// TwinCAT 3 PLC project Plc
// ProgramVersion: 3.1.4023.0
// libraries:
//   Tc2_Standard, * (Beckhoff Automation GmbH)
//   Tc2_System, * (Beckhoff Automation GmbH)
//   Tc3_Module, * (Beckhoff Automation GmbH)
// project tree:
//   / PlcTask.TcTTO (not stored)
//   DUTs/IO/PdoEntries/ Channel_D623F56C.TcDUT
//   DUTs/IO/PDOs/ InfoData_6F19DB2B.TcDUT (not stored), DIG_Outputs_F9744C66.TcDUT, WcState_0B2B16F9.TcDUT, InfoData_32EB74EA.TcDUT, InfoData_E68C61CD.TcDUT (not stored), InfoData_2A97D6CF.TcDUT (not stored), Inputs_A65FACA4.TcDUT (not stored), Outputs_23C0ED1D.TcDUT (not stored)
//   DUTs/IO/Boxes/ EK1100_1FC0878B.TcDUT (not stored), EL2044_DE371F9A.TcDUT
//   DUTs/IO/Devices/ SyncUnitTask_2D604ED5.TcDUT (not stored), SyncUnitTasks_6FEB8257.TcDUT (not stored), SyncUnits_99E584AF.TcDUT (not stored)
//   DUTs/IO/Topology/ Term_1_EK1100_C568EA04.TcDUT (not stored), Device_1_EtherCAT_15E26550.TcDUT (not stored)
//   DUTs/IO/Base/ EtcSlaveBase_82538BE2.TcDUT (not stored), EtcSlaveBase_82538BE2.TcDUT (not stored), EtcSlaveBase_82538BE2.TcDUT (not stored), EtcSlaveTerminalBase_947E5A46.TcDUT (not stored), EtcSlaveBoxBase_77A0E4A7.TcDUT (not stored), EtcSlaveEndTerminalBase_866C7F0C.TcDUT (not stored), InputBase_8311D824.TcDUT (not stored), OutputBase_10CEE7DE.TcDUT (not stored), EtcMasterBase_62654B43.TcDUT (not stored)
//   GVLs/ GVL_iXlinker.TcGVL (not stored)
// real-time tasks:
//   TASK PlcTask: cycle T#10ms, priority 20, ADS port 350
// I/O:
//   DEVICE Device 1 (EtherCAT), AmsNetId 172.20.30.238.2.1
//     Term 1 (EK1100) [EK1100 EtherCAT Coupler (2A E-Bus)]
//       Term 2 (EL2044) [EL2044 4Ch. Dig. Output 24V, 2A, Diagnostic]
// variable links:
//   Plc/Plc Instance <-> Device 1 (EtherCAT)/Term 1 (EK1100)
//     PlcTask Inputs/GVL_iXlinker.Device_1_EtherCAT.Term_1_EK1100.InfoData.State <-> InfoData/State
//   Plc/Plc Instance <-> Device 1 (EtherCAT)/Term 1 (EK1100)/Term 2 (EL2044)
//     PlcTask Outputs/GVL_iXlinker.Device_1_EtherCAT.Term_1_EK1100.Term_2_EL2044.DIG_Outputs.Channel_{1..4}/Output <-> DIG Outputs/Channel {1..4}/Output  (4 links)
//     PlcTask Inputs/GVL_iXlinker.Device_1_EtherCAT.Term_1_EK1100.Term_2_EL2044.WcState.WcState <-> WcState/WcState
//     PlcTask Inputs/GVL_iXlinker.Device_1_EtherCAT.Term_1_EK1100.Term_2_EL2044.InfoData.AdsAddr <-> InfoData/AdsAddr
//     PlcTask Inputs/GVL_iXlinker.Device_1_EtherCAT.Term_1_EK1100.Term_2_EL2044.InfoData.State <-> InfoData/State
//   Plc/Plc Instance <-> Device 1 (EtherCAT)
//     PlcTask Inputs/GVL_iXlinker.Device_1_EtherCAT.SyncUnits._default._unreferenced.WcState.WcState <-> SyncUnits/<default>/<unreferenced>/WcState/WcState
//     PlcTask Inputs/GVL_iXlinker.Device_1_EtherCAT.SyncUnits._default._unreferenced.InfoData.ObjectId <-> SyncUnits/<default>/<unreferenced>/InfoData/ObjectId
//     PlcTask Inputs/GVL_iXlinker.Device_1_EtherCAT.SyncUnits._default._unreferenced.InfoData.State <-> SyncUnits/<default>/<unreferenced>/InfoData/State
//     PlcTask Inputs/GVL_iXlinker.Device_1_EtherCAT.SyncUnits._default._unreferenced.InfoData.SlaveCount <-> SyncUnits/<default>/<unreferenced>/InfoData/SlaveCount
//     PlcTask Inputs/GVL_iXlinker.Device_1_EtherCAT.SyncUnits._default.PlcTask.WcState.WcState <-> SyncUnits/<default>/PlcTask/WcState/WcState
//     PlcTask Inputs/GVL_iXlinker.Device_1_EtherCAT.SyncUnits._default.PlcTask.InfoData.ObjectId <-> SyncUnits/<default>/PlcTask/InfoData/ObjectId
//     PlcTask Inputs/GVL_iXlinker.Device_1_EtherCAT.SyncUnits._default.PlcTask.InfoData.State <-> SyncUnits/<default>/PlcTask/InfoData/State
//     PlcTask Inputs/GVL_iXlinker.Device_1_EtherCAT.SyncUnits._default.PlcTask.InfoData.SlaveCount <-> SyncUnits/<default>/PlcTask/InfoData/SlaveCount
//     PlcTask Inputs/GVL_iXlinker.Device_1_EtherCAT.Inputs.SlaveCount <-> Inputs/SlaveCount
//     PlcTask Inputs/GVL_iXlinker.Device_1_EtherCAT.Inputs.DevState <-> Inputs/DevState
//     PlcTask Inputs/GVL_iXlinker.Device_1_EtherCAT.Inputs.Frm0State <-> Inputs/Frm0State
//     PlcTask Inputs/GVL_iXlinker.Device_1_EtherCAT.Inputs.Frm0WcState <-> Inputs/Frm0WcState
//     PlcTask Inputs/GVL_iXlinker.Device_1_EtherCAT.Inputs.Frm0InputToggle <-> Inputs/Frm0InputToggle
//     PlcTask Outputs/GVL_iXlinker.Device_1_EtherCAT.Outputs.DevCtrl <-> Outputs/DevCtrl
//     PlcTask Outputs/GVL_iXlinker.Device_1_EtherCAT.Outputs.Frm0Ctrl <-> Outputs/Frm0Ctrl
//     PlcTask Outputs/GVL_iXlinker.Device_1_EtherCAT.Outputs.Frm0WcCtrl <-> Outputs/Frm0WcCtrl
//     PlcTask Inputs/GVL_iXlinker.Device_1_EtherCAT.InfoData.ChangeCount <-> InfoData/ChangeCount
//     PlcTask Inputs/GVL_iXlinker.Device_1_EtherCAT.InfoData.DevId <-> InfoData/DevId
//     PlcTask Inputs/GVL_iXlinker.Device_1_EtherCAT.InfoData.AmsNetId <-> InfoData/AmsNetId
//     PlcTask Inputs/GVL_iXlinker.Device_1_EtherCAT.InfoData.CfgSlaveCount <-> InfoData/CfgSlaveCount
//     PlcTask Inputs/GVL_iXlinker.Device_1_EtherCAT.InfoData.DcToTcTimeOffset <-> InfoData/DcToTcTimeOffset
//     PlcTask Inputs/GVL_iXlinker.Device_1_EtherCAT.InfoData.DcToExtTimeOffset <-> InfoData/DcToExtTimeOffset

// ---- DUTs/IO/PdoEntries/Channel_D623F56C.TcDUT
{attribute 'GeneratedUsingTerminal: EL2044-0000-0016'}
{attribute addProperty BoxType "EL2044-0000-0016"}
{attribute addProperty Id "OutputBOOL1"}
{attribute addProperty CRC "3592680812"}
{attribute addProperty Size "1"}
TYPE Channel_D623F56C :
STRUCT
	{attribute addProperty Name "Output"}
	Output : BOOL;
END_STRUCT
END_TYPE

// ---- DUTs/IO/PDOs/DIG_Outputs_F9744C66.TcDUT
{attribute 'GeneratedUsingTerminal: EL2044-0000-0016'}
{attribute addProperty BoxType "EL2044-0000-0016"}
{attribute addProperty Id "Channel_1AT %Q*Channel_D623F56C1Channel_2AT %Q*Channel_D623F56C1Channel_3AT %Q*Channel_D623F56C1Channel_4AT %Q*Channel_D623F56C1"}
{attribute addProperty CRC "4185148518"}
{attribute addProperty Size "4"}
TYPE DIG_Outputs_F9744C66 EXTENDS OutputBase_10CEE7DE :
STRUCT
	{attribute addProperty Name "Channel_1"}
	Channel_1 AT %Q* : Channel_D623F56C;
	{attribute addProperty Name "Channel_2"}
	Channel_2 AT %Q* : Channel_D623F56C;
	{attribute addProperty Name "Channel_3"}
	Channel_3 AT %Q* : Channel_D623F56C;
	{attribute addProperty Name "Channel_4"}
	Channel_4 AT %Q* : Channel_D623F56C;
END_STRUCT
END_TYPE

// ---- DUTs/IO/PDOs/WcState_0B2B16F9.TcDUT
{attribute 'GeneratedUsingTerminal: EL2044-0000-0016'}
{attribute addProperty BoxType "EL2044-0000-0016"}
{attribute addProperty Id "WcStateAT %I*BOOL1"}
{attribute addProperty CRC "187373305"}
{attribute addProperty Size "1"}
TYPE WcState_0B2B16F9 :
STRUCT
	{attribute addProperty Name "WcState"}
	WcState AT %I* : BOOL;
END_STRUCT
END_TYPE

// ---- DUTs/IO/PDOs/InfoData_32EB74EA.TcDUT
{attribute 'GeneratedUsingTerminal: EL2044-0000-0016'}
{attribute addProperty BoxType "EL2044-0000-0016"}
{attribute addProperty Id "AdsAddrAT %I*AMSADDR8StateAT %I*UINT2"}
{attribute addProperty CRC "854291690"}
{attribute addProperty Size "10"}
TYPE InfoData_32EB74EA EXTENDS InputBase_8311D824 :
STRUCT
	{attribute addProperty Name "AdsAddr"}
	AdsAddr AT %I* : AMSADDR;
	{attribute addProperty Name "State"}
	State AT %I* : UINT;
END_STRUCT
END_TYPE

// ---- DUTs/IO/Boxes/EL2044_DE371F9A.TcDUT
{attribute 'GeneratedUsingTerminal: EL2044-0000-0016'}
{attribute addProperty BoxType "EL2044-0000-0016"}
{attribute addProperty Description "EL2044 4Ch. Dig. Output 24V, 2A, Diagnostic"}
{attribute addProperty Physics "KK"}
{attribute addProperty Id "DIG_OutputsAT %Q*DIG_Outputs_F9744C664WcStateAT %I*WcState_0B2B16F91InfoDataAT %I*InfoData_32EB74EA10"}
{attribute addProperty CRC "3728154522"}
{attribute addProperty Size "15"}
TYPE EL2044_DE371F9A EXTENDS EtcSlaveTerminalBase_947E5A46 :
STRUCT
	{attribute addProperty Name "DIG_Outputs"}
	DIG_Outputs : DIG_Outputs_F9744C66;
	{attribute addProperty Name "WcState"}
	WcState : WcState_0B2B16F9;
	{attribute addProperty Name "InfoData"}
	InfoData : InfoData_32EB74EA;
END_STRUCT
END_TYPE
